PROGRAM MAIN
VAR
	fbUnit : FB_Unit;
	fbLogger : FB_Logger;
END_VAR

fbUnit.Initalize(fbLogger);
fbUnit();

fbLogger.Write('C:/Test.csv');

END_PROGRAM

(* stored: Version 1.1.0.1, ProductVersion 3.1.4024.12
   POU MAIN: Id {4df7eff0-0a82-4582-95f2-d69fae3df5f6}, SpecialFunc None *)
